FUNCTION_BLOCK "Convention66"
TITLE = "% VERSION:      Q       1.4 %" # Violation
BEGIN
END_FUNCTION_BLOCK
